{attribute addProperty BoxType "EL6614-0000-0016"}
{attribute addProperty Id "InfoDataInfoData_BC63D37F8010"}
{attribute addProperty CRC "424293389"}
{attribute addProperty SizeInBites "80"}
{attribute addProperty SizeInBytes "10"}
TYPE EL6614_194A340D :
STRUCT
	{attribute addProperty Name "InfoData"}
	InfoData : InfoData_BC63D37F;
END_STRUCT
END_TYPE

(* stored: Version 1.2.0.0, ProductVersion 3.1.4024.9
   DUT EL6614_194A340D: Id {8a0b8d84-69a4-4deb-999e-f7215db134c3} *)
